PROGRAM ups_CX51X0
VAR_INPUT
	bWrtie					: BOOL;//触发保存
END_VAR
VAR
	//fbUPS					: FB_S_UPS;
	fbUPS					: FB_S_UPS_CX51x0;
	fbGetCurTaskIndex		: GetCurTaskIndex;
	fbWritePersistentData	: FB_WritePersistentData;
	nTaskNo					: INT;
	wrtieR_TRIG				: R_TRIG;
END_VAR

(* 需要在变量改变之后, PLC断电之前触发bWrtie *)
wrtieR_TRIG(CLK:=bWrtie);

fbGetCurTaskIndex(index=>nTaskNo);
fbWritePersistentData(
	NETID:= , 
	PORT:= 851, 
	START:= wrtieR_TRIG.Q OR TwinCAT_SystemInfoVarList._TaskInfo[nTaskNo].FirstCycle, 
	TMOUT:= , 
	MODE:= , 
	BUSY=> , 
	ERR=> , 
	ERRID=> );

IF wrtieR_TRIG.Q THEN
	bWrtie:=FALSE;
END_IF

(* 以下仅用于带1s UPS的CX51x0 PLC *)
fbUPS(
	sNetID:= , 
	iPLCPort:= 851, 
	iUPSPort:= , 
	tTimeout:= , 
	eUpsMode:= , 
	ePersistentMode:= , 
	tRecoverTime:= , 
	bPowerFailDetect=> , 
	eState=> );

METHOD Act_Wrtie
VAR_INPUT
END_VAR
bWrtie:=TRUE;
END_METHOD

ACTION VersionLog:
(*
版本: V1.0.0.0
说明:
	1. 首个版本
(**************************************************)
版本: V1.0.0.1
说明:
	1. 修正断电保持失效功能
(**************************************************)
版本: V1.0.0.2
说明:
	1. 怎么函数Act_Wrtie()，方便外部调用
(**************************************************)
*)
END_ACTION

END_PROGRAM

(* stored: Version 1.1.0.1, ProductVersion 3.1.4024.4
   POU ups_CX51X0: Id {4f96daf2-9a58-4919-b377-4ed8dbb71b97}, SpecialFunc None
   Method Act_Wrtie: Id {2e2e1f6e-2e73-4aef-85ef-84f729a57cac}
   Action VersionLog: Id {d788d662-c585-4bd2-9e14-df91bb62f382} *)
